// TIA Portal V18 export
TYPE "TM_Count_Man_In"
   STRUCT
      COUNT_VALUE : DInt;
      CAPTURED_VALUE : DInt;
      MEASURED_VALUE : DInt;
      POWER_ERROR : Bool;
      ENC_ERROR : Bool;
      LD_ERROR : Bool;
      Reserved1 : Bool;
      Reserved2 : Bool;
      Reserved3 : Bool;
      Reserved4 : Bool;
      Reserved5 : Bool;
      Reserved6 : Bool;
      RES_EVENT_ACK : Bool;
      LD_STS_SLOT0 : Bool;
      LD_STS_SLOT1 : Bool;
      STS_READY : Bool;
      STS_SW_GATE : Bool;
      Reserved7 : Bool;
      Reserved8 : Bool;
      STS_DIR : Bool;
      STS_CNT : Bool;
      STS_GATE : Bool;
      STS_DQ0 : Bool;
      STS_DQ1 : Bool;
      STS_DI0 : Bool;
      STS_DI1 : Bool;
      STS_DI2 : Bool;
      EVENT_ZERO : Bool;
      EVENT_UFLW : Bool;
      EVENT_OFLW : Bool;
      EVENT_CMP0 : Bool;
      EVENT_CMP1 : Bool;
      EVENT_SYNC : Bool;
      EVENT_CAP : Bool;
      STS_M_INTERVAL : Bool;
   END_STRUCT;
END_TYPE
